TYPE ST_SafetyFunctionOut :
STRUCT
    byRaw : BYTE;
END_STRUCT
END_TYPE

(* stored: Version 1.1.0.1
   DUT ST_SafetyFunctionOut: Id {d225f0e9-f4be-0268-2036-d232ca0275b9} *)
